Omron Sysmac Studio project AcceptTCPReceiveTCPSendTCP (Sysmac Studio 1.56.0.64011, StandardProject)

# Controller HCS_Etch: NJ501-1300 version 1.18
Units and slaves: Power Supply : NJ-Px3001; CPU : NJ501-1300
Task PrimaryTask (priority 4, period or condition 1000): Program0

VAR_GLOBAL
    SKTPressme : BOOL;
    SKT_busy : BOOL;
    SKT_error : BOOL;
    SKT_errorID : WORD;
    SKTSKT : _sSOCKET;
    SendSKTDat : ARRAY[0..1999] of BYTE;
    SKTtcpCbusy : BOOL;
    SKTtcpCerror : BOOL;
    SKTtcpCerrorID : WORD;
    SKTclearBbusy : BOOL;
    SKTclearBerror : BOOL;
    SKTclearBerrorID : WORD;
    AcceptPress : BOOL;
    SendSKTDatString : STRING[255];
    SKTDataString : STRING[255] := 'ABC';
    def : UINT;
    RCVDataString : STRING[256] := 'ABC Received';
    closeSKTSKT2 : BOOL;
END_VAR

PROGRAM Program0
VAR
    ConnectSKT : SktTCPConnect;
    AcceptSKT : SktTCPAccept;
    ClearBuff : SktClearBuf;
    SendSKT : SktTCPSend;
    CloseSKT : SktClose;
    closeSKTSKT : BOOL;
    SendME : BOOL;
    SKTtcpSbusy : BOOL;
    SKTtcpSerror : BOOL;
    SKTtcpSerrorID : WORD;
    ReceiveSENT : BOOL;
    ReceiveSKT : SktTCPRcv;
    SKTtcpRerrorID : WORD;
    SKTtcpRerror : BOOL;
    SKTtcpRbusy : BOOL;
    SKTSendDat : ARRAY[0..1999] of BYTE := [2000(16#0)];
    SKTRcvDat : Array[0..1999] of BYTE := [2000(16#0)];
    SKTSKT1 : _sSOCKET := (Handle:=0, SrcAdr:=(PortNo:=0, IpAdr:=''), DstAdr:=(PortNo:=0, IpAdr:=''));
    GetTCPStatus : SktGetTCPStatus;
    SKTgettcpSbusy : BOOL;
    SKTgettcpSerror : BOOL;
    SKTgettcpSerrorID : WORD;
    Clearpress : BOOL;
    Sendpress : BOOL;
    abclen : UINT;
    Byteabc : UINT;
    deflen : UINT;
    RCVDataString : STRING[256] := '_ACK';
    Bytedef : BOOL;
    SendReceivedmsg : SktTCPSend;
    BusyR : BOOL;
    ErrorR : BOOL;
    ErrorIDR : WORD;
    SendFinish : BOOL;
    Clearbufbool : BOOL;
    GetStatus : BOOL;
    StatusTCP : _eCONNECTION_STATE;
    SKTReceiveDat : ARRAY[0..1999] OF BYTE := [2000(16#0)];
    Bytdef : UINT;
    SKTtcpSendReceiveB : BOOL;
    SKTtcpSendReceiveE : BOOL;
    SKTtcpSendReceiveEID : WORD;
    SKTReceiveSize : UINT;
    ReceiveFlagDat : BOOL;
    CStatus : STRING[256] := 'ESTABLISHED';
    SKTtcpAbusy : BOOL;
    SKTtcpAerror : BOOL;
    SKTtcpAerrorID : WORD;
    SKTTrigger : BOOL;
    defbye : UINT;
    defbyte : UINT;
    GetStatus2 : BOOL;
    Sendpress2 : BOOL;
    ReceiveFlagDat2 : BOOL;
    ReceiveSKT2 : SktTCPRcv;
    SendReceivedmsg2 : SktTCPSend;
    CloseSKT2 : SktClose;
    GetTCPStatus2 : SktGetTCPStatus;
    SendSKT2 : SktTCPSend;
END_VAR
VAR_EXTERNAL
    SKTPressme : BOOL;
    SKT_busy : BOOL;
    SKT_error : BOOL;
    SKT_errorID : WORD;
    SKTSKT : _sSOCKET;
    SendSKTDat : ARRAY[0..1999] of BYTE;
    SKTtcpCbusy : BOOL;
    SKTtcpCerror : BOOL;
    SKTtcpCerrorID : WORD;
    SKTclearBbusy : BOOL;
    SKTclearBerror : BOOL;
    SKTclearBerrorID : WORD;
    AcceptPress : BOOL;
    SendSKTDatString : STRING[255];
    SKTDataString : STRING[255];
    def : UINT;
    closeSKTSKT2 : BOOL;
END_VAR

(* Section Section0: ladder, written here as Structured Text *)

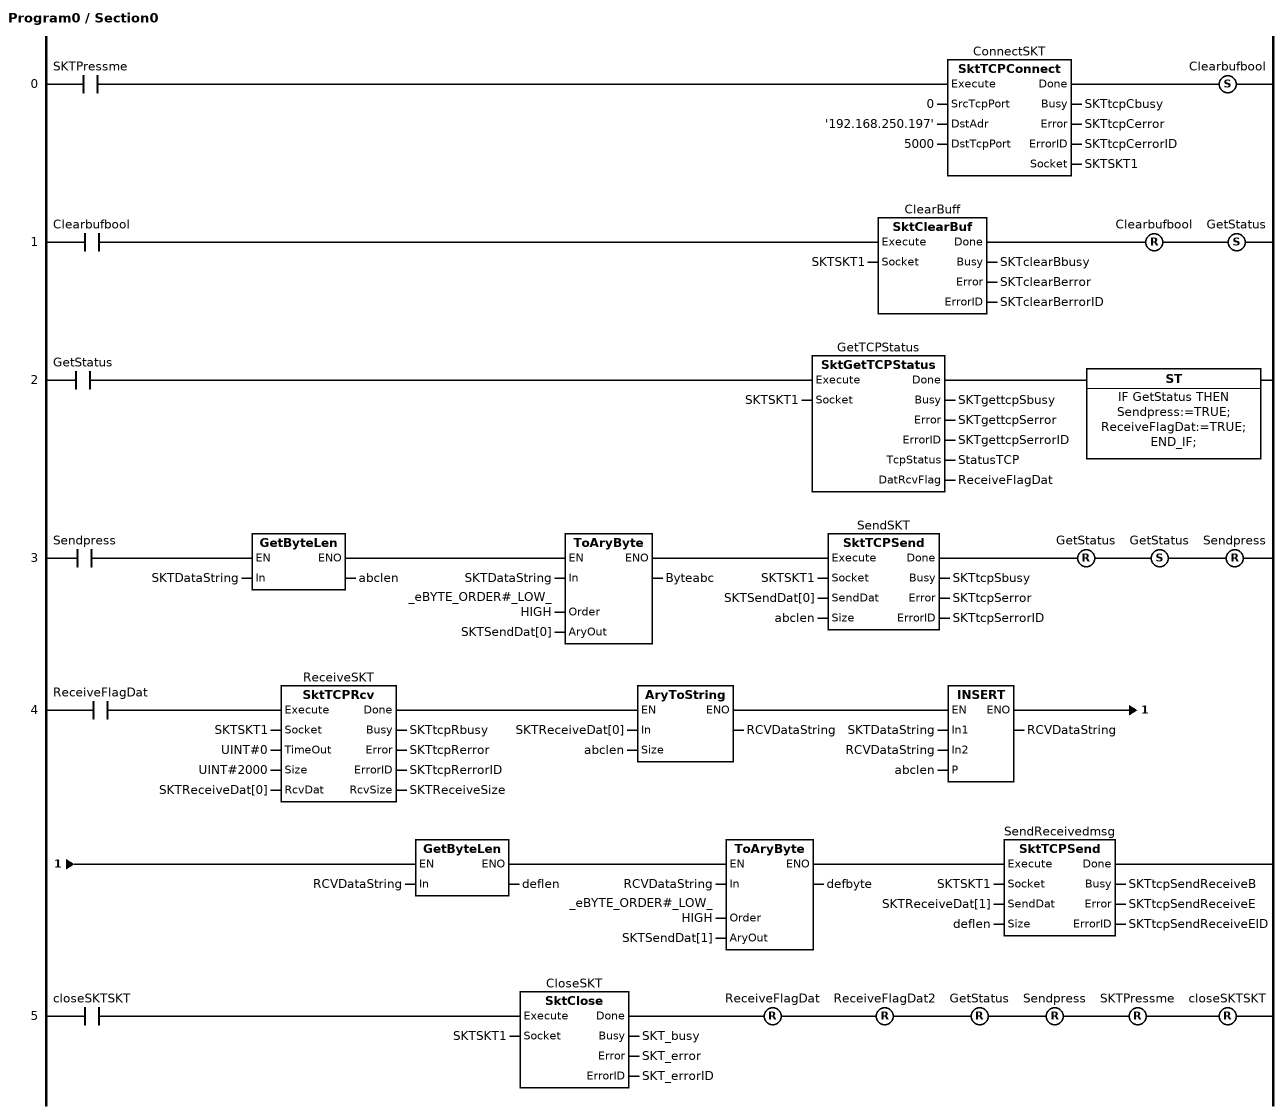
(* Rung 0 *)
ConnectSKT(Execute := SKTPressme, SrcTcpPort := 0, DstAdr := '192.168.250.197', DstTcpPort := 5000, Busy => SKTtcpCbusy, Error => SKTtcpCerror, ErrorID => SKTtcpCerrorID, Socket => SKTSKT1);
IF ConnectSKT.Done THEN Clearbufbool := TRUE; END_IF;
(* Rung 1 *)
ClearBuff(Execute := Clearbufbool, Socket := SKTSKT1, Busy => SKTclearBbusy, Error => SKTclearBerror, ErrorID => SKTclearBerrorID);
IF ClearBuff.Done THEN
    Clearbufbool := FALSE;
    GetStatus := TRUE;
END_IF;
(* Rung 2 *)
GetTCPStatus(Execute := GetStatus, Socket := SKTSKT1, Busy => SKTgettcpSbusy, Error => SKTgettcpSerror, ErrorID => SKTgettcpSerrorID, TcpStatus => StatusTCP, DatRcvFlag => ReceiveFlagDat);
IF GetTCPStatus.Done THEN
    IF GetStatus THEN
    	Sendpress:=TRUE;
    	ReceiveFlagDat:=TRUE;
    END_IF;
    
    	
END_IF;
(* Rung 3 *)
IF Sendpress THEN
    abclen := GetByteLen(In := SKTDataString);
    Byteabc := ToAryByte(In := SKTDataString, Order := _eBYTE_ORDER#_LOW_HIGH, AryOut := SKTSendDat[0]);
END_IF;
SendSKT(Execute := Sendpress, Socket := SKTSKT1, SendDat := SKTSendDat[0], Size := abclen, Busy => SKTtcpSbusy, Error => SKTtcpSerror, ErrorID => SKTtcpSerrorID);
IF SendSKT.Done THEN
    GetStatus := FALSE;
    GetStatus := TRUE;
    Sendpress := FALSE;
END_IF;
(* Rung 4 *)
ReceiveSKT(Execute := ReceiveFlagDat, Socket := SKTSKT1, TimeOut := UINT#0, Size := UINT#2000, RcvDat := SKTReceiveDat[0], Busy => SKTtcpRbusy, Error => SKTtcpRerror, ErrorID => SKTtcpRerrorID, RcvSize => SKTReceiveSize);
IF ReceiveSKT.Done THEN
    RCVDataString := AryToString(In := SKTReceiveDat[0], Size := abclen);
    RCVDataString := INSERT(In1 := SKTDataString, In2 := RCVDataString, P := abclen);
    deflen := GetByteLen(In := RCVDataString);
    defbyte := ToAryByte(In := RCVDataString, Order := _eBYTE_ORDER#_LOW_HIGH, AryOut := SKTSendDat[1]);
END_IF;
SendReceivedmsg(Execute := ReceiveSKT.Done, Socket := SKTSKT1, SendDat := SKTReceiveDat[1], Size := deflen, Busy => SKTtcpSendReceiveB, Error => SKTtcpSendReceiveE, ErrorID => SKTtcpSendReceiveEID);
(* Rung 5 *)
CloseSKT(Execute := closeSKTSKT, Socket := SKTSKT1, Busy => SKT_busy, Error => SKT_error, ErrorID => SKT_errorID);
IF CloseSKT.Done THEN
    ReceiveFlagDat := FALSE;
    ReceiveFlagDat2 := FALSE;
    GetStatus := FALSE;
    Sendpress := FALSE;
    SKTPressme := FALSE;
    closeSKTSKT := FALSE;
END_IF;

(* Section Section1: ladder, written here as Structured Text *)

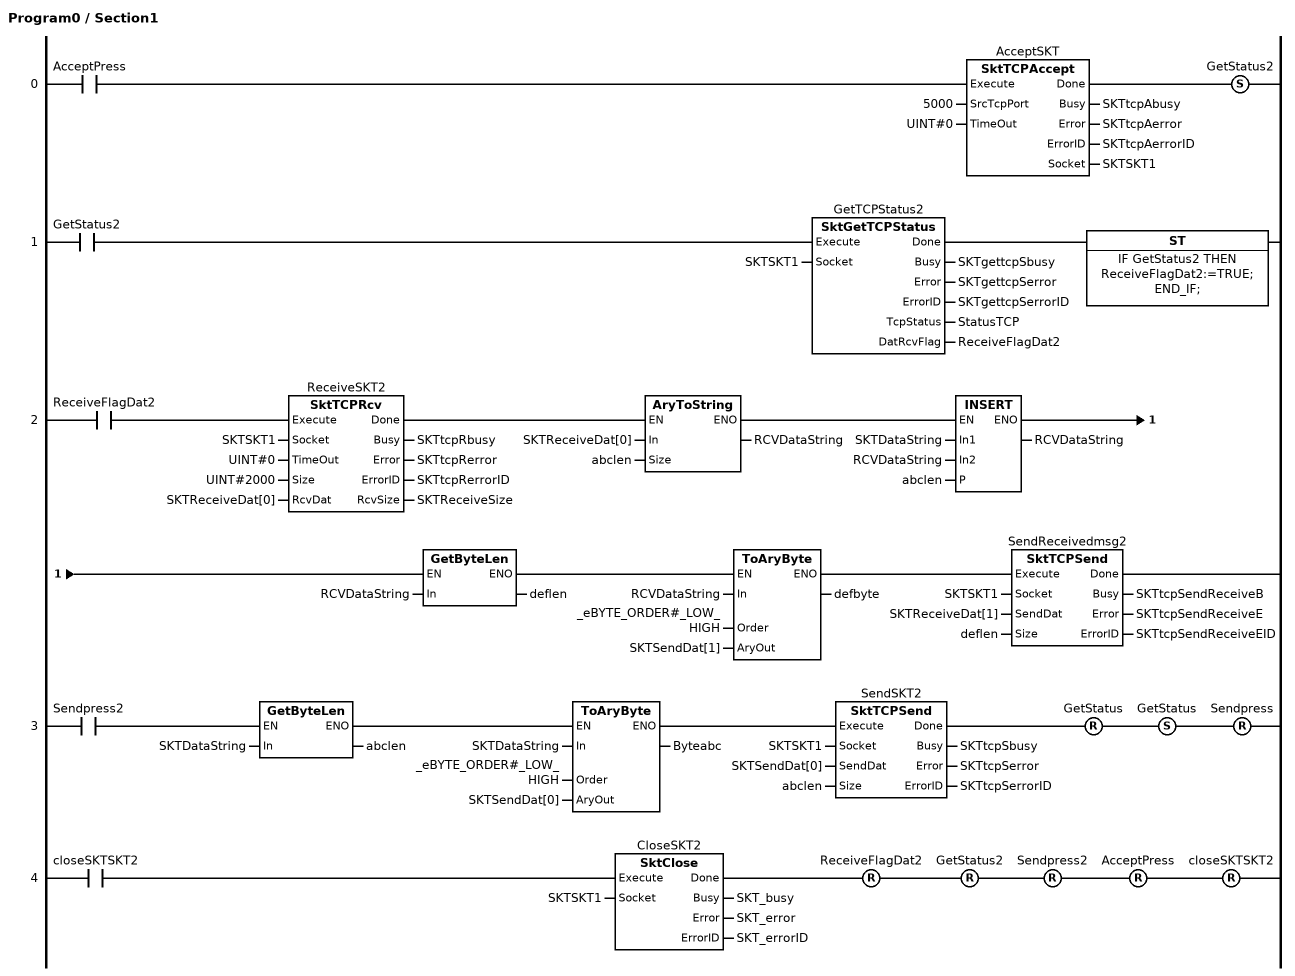
(* Rung 0 *)
AcceptSKT(Execute := AcceptPress, SrcTcpPort := 5000, TimeOut := UINT#0, Busy => SKTtcpAbusy, Error => SKTtcpAerror, ErrorID => SKTtcpAerrorID, Socket => SKTSKT1);
IF AcceptSKT.Done THEN GetStatus2 := TRUE; END_IF;
(* Rung 1 *)
GetTCPStatus2(Execute := GetStatus2, Socket := SKTSKT1, Busy => SKTgettcpSbusy, Error => SKTgettcpSerror, ErrorID => SKTgettcpSerrorID, TcpStatus => StatusTCP, DatRcvFlag => ReceiveFlagDat2);
IF GetTCPStatus2.Done THEN
    IF GetStatus2 THEN
    	ReceiveFlagDat2:=TRUE;
    END_IF;
    
    	
END_IF;
(* Rung 2 *)
ReceiveSKT2(Execute := ReceiveFlagDat2, Socket := SKTSKT1, TimeOut := UINT#0, Size := UINT#2000, RcvDat := SKTReceiveDat[0], Busy => SKTtcpRbusy, Error => SKTtcpRerror, ErrorID => SKTtcpRerrorID, RcvSize => SKTReceiveSize);
IF ReceiveSKT2.Done THEN
    RCVDataString := AryToString(In := SKTReceiveDat[0], Size := abclen);
    RCVDataString := INSERT(In1 := SKTDataString, In2 := RCVDataString, P := abclen);
    deflen := GetByteLen(In := RCVDataString);
    defbyte := ToAryByte(In := RCVDataString, Order := _eBYTE_ORDER#_LOW_HIGH, AryOut := SKTSendDat[1]);
END_IF;
SendReceivedmsg2(Execute := ReceiveSKT2.Done, Socket := SKTSKT1, SendDat := SKTReceiveDat[1], Size := deflen, Busy => SKTtcpSendReceiveB, Error => SKTtcpSendReceiveE, ErrorID => SKTtcpSendReceiveEID);
(* Rung 3 *)
IF Sendpress2 THEN
    abclen := GetByteLen(In := SKTDataString);
    Byteabc := ToAryByte(In := SKTDataString, Order := _eBYTE_ORDER#_LOW_HIGH, AryOut := SKTSendDat[0]);
END_IF;
SendSKT2(Execute := Sendpress2, Socket := SKTSKT1, SendDat := SKTSendDat[0], Size := abclen, Busy => SKTtcpSbusy, Error => SKTtcpSerror, ErrorID => SKTtcpSerrorID);
IF SendSKT2.Done THEN
    GetStatus := FALSE;
    GetStatus := TRUE;
    Sendpress := FALSE;
END_IF;
(* Rung 4 *)
CloseSKT2(Execute := closeSKTSKT2, Socket := SKTSKT1, Busy => SKT_busy, Error => SKT_error, ErrorID => SKT_errorID);
IF CloseSKT2.Done THEN
    ReceiveFlagDat2 := FALSE;
    GetStatus2 := FALSE;
    Sendpress2 := FALSE;
    AcceptPress := FALSE;
    closeSKTSKT2 := FALSE;
END_IF;
END_PROGRAM